# EPICS autosave request: iocBoot/generic_motors_ioc/dbSave/DAC128_single.req
%
% BURT Request File
%
% Single channel DAC128 saved
%

$(P)DAC$(D)_$(N)_tweakVal.VAL

$(P)DAC$(D)_$(N).EGUL
$(P)DAC$(D)_$(N).DRVL
$(P)DAC$(D)_$(N).LOPR

$(P)DAC$(D)_$(N).EGUF
$(P)DAC$(D)_$(N).DRVH
$(P)DAC$(D)_$(N).HOPR

% $(P)DAC$(D)_$(N).VAL
% $(P)DAC$(D)_$(N)_pulse.VAL
